// TwinCAT 3 PLC project TestCode
// ProgramVersion: 3.1.4022.3
// libraries:
//   Tc2_Standard, * (Beckhoff Automation GmbH)
//   Tc2_System, * (Beckhoff Automation GmbH)
//   Tc3_Module, * (Beckhoff Automation GmbH)
// project tree:
//   GVLs/ VARS.TcGVL
//   / PlcTask.TcTTO (not stored)
//   POUs/ MAIN.TcPOU
// real-time tasks:
//   TASK PlcTask: cycle T#10ms, priority 4, ADS port 350
// I/O:
//   DEVICE Device 1 (EtherCAT), AmsNetId 5.49.22.42.2.1
//     Term 4 (EK1200) [EK1200-5000 EtherCAT Power supply (2A E-Bus)]
//       Term 5 (EL5101) [EL5101 1Ch. Inc. Encoder 5V]
//       Term 6 (EL1008) [EL1008 8Ch. Dig. Input 24V, 3ms]
//       Term 7 (EL2008) [EL2008 8Ch. Dig. Output 24V, 0.5A]
//       Term 8 (EL9011) [EL9011 End Terminal]
//   DEVICE Device 4 (COM Port)
// variable links:
//   TestCode/TestCode Instance <-> Device 1 (EtherCAT)/Term 4 (EK1200)/Term 7 (EL2008)
//     PlcTask Outputs/MAIN.out1 <-> Channel 1/Output

// ---- GVLs/VARS.TcGVL
{attribute 'qualified_only'}
VAR_GLOBAL
	iTest1 	: UINT; (*~ (OPC: 1 : available for OPC-clients) 
					(OPC_PROP[0005]: 3 : OPC_PROP_RIGHTS, here read/write) *)
	iTest2 	: UINT;	(*~ (OPC: 1 : available for OPC-clients) *)
	iSum 	: UINT; (*~ (OPC: 1 : available for OPC-clients) 
					(OPC_PROP[0005]: 1 : OPC_PROP_RIGHTS, here read only) *)
END_VAR

// ---- POUs/MAIN.TcPOU
PROGRAM MAIN
VAR
	heartbeat : BYTE;
	out1 AT %Q* : BOOL;
	outVal1 : BOOL;
END_VAR

VARS.iSum := VARS.iTest1 + VARS.iTest2 + 10;
//heartbeat:= heartbeat+1;
out1 := outval1;

END_PROGRAM
